FUNCTION_BLOCK FB_SendDriveReset_1
VAR_INPUT
	DriveReset : INT;
END_VAR
VAR_OUTPUT
END_VAR
VAR
	TxMessage : EXTCANQUEUE;
END_VAR
VAR_IN_OUT
	CAN_OUTPUTS_1 : CANTXQUEUESTRUCT_E_32;
	CAN_INPUTS_1 : CANRXQUEUESTRUCT_E_32;
END_VAR

 
TxMessage.cobId := 150;
TxMessage.length := 1;
TxMessage.data[0] :=  INT_TO_BYTE(DriveReset AND 16#FF);
CAN_OUTPUTS_1.TxMessages[8] := TxMessage;
//CAN_OUTPUTS.NoOfTxMessages := 1;

(*
TxMessage.cobId := 120;
TxMessage.length := 1;
TxMessage.data[0] :=  INT_TO_BYTE(PropFlag AND 16#FF);
CAN_OUTPUTS.TxMessages[5] := TxMessage;
CAN_OUTPUTS.TxCounter := CAN_INPUTS.TxCounter + 1;
*)

END_FUNCTION_BLOCK

(* stored: Version 1.1.0.1
   POU FB_SendDriveReset_1: Id {d43fc5b7-a1a3-4570-bd9a-76a1b8f88161}, SpecialFunc None *)
